FUNCTION DivisionFunction : REAL
VAR_INPUT
	i_rValueA : REAL;
	i_rValueB : REAL;
END_VAR
VAR
END_VAR

IF	i_rValueB <> 0 THEN
DivisionFunction := i_rValueA / i_rValueB;
ELSE
	DivisionFunction := 0;
END_IF

END_FUNCTION

(* stored: Version 1.1.0.1, ProductVersion 3.1.4022.12
   POU DivisionFunction: Id {900c89e1-6993-478e-b002-c5f5cf93cd4b}, SpecialFunc None *)
